// TIA Portal project "Project_MQTT" (V15.1)

(* hardware
DEVICE "S71500/ET200MP station_1"  S7-1500 station
   slot 0: "Rail_0"  Rack  6ES7 590-1***0-0AA0
   slot 1: "PLC_1"  CPU 1516F-3 PN/DP  6ES7 516-3FN01-0AB0  V2.6
      slot 3: "CPU display_1"  6ES7591-1BA00-0AA0
   slot 2: "TM Count 2x24V_1"  TM Count 2x24V  6ES7 550-1AA00-0AB0  V1.3
*)

// ===== PLC "PLC_1"  CPU 1516F-3 PN/DP =====

VAR_GLOBAL   // PLC tag table "Default tag table"
   "mxEnable" AT %M0.0 : Bool;
   "mxSaveIntoBroker" AT %M0.1 : Bool;
   "mxsubscribe" AT %M0.2 : Bool;
   "mxunsubscribe" AT %M0.3 : Bool;
   "mxPublishData" AT %M0.4 : Bool;
   "mxPublishData1" AT %M0.5 : Bool;
   "mxPublishData2" AT %M0.6 : Bool;
   "mxdone" AT %M0.7 : Bool;
   "Tag_1" AT %MW100 : Int;
END_VAR

// folder: 02_Types/S7-1500

TYPE "LMQTT_typePublishData"
   STRUCT
      publishMessage : Bool;   // Set to true. Can be reset to false once done flag is set be FB
      publishTopic : WString[250];   // Size be increased, but must increase MAX_SENDBUFFER and MAX_PUBLISH_MESSAGE in the FB
      publishMessageData : WString[1500];   // Size be increased, but must increase MAX_SENDBUFFER and MAX_PUBLISH_MESSAGE in the FB
      publishQoS : Int;   // Defines the QoS level for the MQTT message. 0,1 and 2 supported
      publishRetainFlag : Bool;   // If true, message may be saved at the broker
   END_STRUCT;
END_TYPE

TYPE "LMQTT_typeSubscribeData"
   STRUCT
      subscribeToTopic : Bool;   // When true, subscribes to the topic indicated by "subscriptionTopic"
      unsubscribeFromTopic : Bool;   // When true, unsubscribes from the "subscriptionTopic"
      subscriptionTopic : WString[250];   // Topic name to subscribe to or unsubscribe off
      subscriptionQoS : Int;   // Defines the QoS level for the MQTT message at the subscriber side. 0 and 1 allowed
   END_STRUCT;
END_TYPE

TYPE "LMQTT_typeSubscriptionData"
   STRUCT
      newMessageRecieved : Bool;   // Is TRUE for one cycle to signal that new data was recieved
      messageInvalid : Bool;   // Is TRUE, when either internal Buffer of FB is too small or recieved Message Data string length is too low
      receivingTopic : WString[400];   // The topic for which the message was recieved
      receivedMessageData : WString[2400];   // The received data (payload)
   END_STRUCT;
END_TYPE

TYPE "LMQTT_typeTcpConnParamData"
   STRUCT
      useQdn : Bool;   // When TRUE, configure the connection for TCP over the fully qualified domain name
      hwIdentifier : Hw_Any;   // HW_ID of the PROFINET interface of the CPU
      connectionID : Conn_Ouc;   // ID of the TCP connection
      qdnAdressBroker : String[254];   // URL of the MQTT Broker . Must end with a dot (".")
      ipAdressBroker : Array[0..3] of USInt;   // IP Address of the broker, e.g.: for the address "192.168.0.10"
      localPort : UInt := 0;   // Local port number of the CPU
      mqttPort : UInt := 1884;   // Remote port of the MQTT broker
      activateSecureConn : Bool;   // When TRUE, the communication is secured via TLS
      validateSubjectAlternateNameOfServer : Bool;   // Only relevant for Client side. If set to True, Client will validate IP address of broker against SAN in the certificate of the MQTT broker
      idTlsServerCertificate : UDInt;   // Identifier of X.509 certificate (usually a CA certificate) to validate the authetication of the TLS server. Only relevant, if "activateSecureConn" is "true"
      idTlsOwnCertificate : UDInt;   // Identifier of own X.509 certificate to validate the own authetication against the TLS server. Only relevant, if "activateSecureConn" is "true" and the TLS server requests a client authentication
   END_STRUCT;
   // // ipAdressBroker[0] : "192"
   // // ipAdressBroker[1] : "168"
   // // ipAdressBroker[2] : "0"
   // // ipAdressBroker[3] : "10"
END_TYPE

TYPE "LMQTT_typeParamData"
   STRUCT
      connectFlag : "LMQTT_typeConnectFlags";
      keepAlive : UInt := 30;   // can be set to higher or lower time // Default is 60 Seconds / KeepAlive in Seconds. 0=No Keepalive
      clientIdentifier : String[23] := 'Siemens SIMATIC';   // should be PROFINET devicename / Unique name of the client used from the client to identify itself at the broker during the connection establishment
      willTopic : String[100];   // specify topic where to send last will / If the will flag is set, the topic for the last will need to be defined
      willMessage : String[100];   // specify last will message which can be sent, see connect flags / If the will flag is set, the message for the last will needs to be defined
      userName : String[100];   // must be set, if flag "username" is true / If the username flag is set, the username for the login at the broker needs to be defined
      password : String[200];   // must be set, if flag "password" is true / If the password flag is set, the password for the login at the broker needs to be defined
   END_STRUCT;
END_TYPE

TYPE "LMQTT_typeConnectFlags"
   STRUCT
      cleanSession : Bool;   // if true, MQTT will create a clean Session at the Broker / When TRUE, all data from a previous session will be deleted
      will : Bool;   // if True, a last Will is sent when Mqtt Client (PLC) disconnects Broker / When TRUE, activates the last will and testament function
      willQoS1 : Bool;   // true, if QoS = 1 / When TRUE, the QoS has level 1 for the last will
      willQoS2 : Bool;   // true, if QoS = 2 / When TRUE, the QoS has level 2 for the last will
      willRetain : Bool;   // must be false, if Will flag is false / When TRUE, the last will is stored at the broker after its been sent
      password : Bool;   // if true, a password is required / When TRUE, the MQTT broker requires a login (name and password) of the client
      userName : Bool;   // if true, a username is required / When TRUE, the MQTT broker requires a login (name and password) of the client
   END_STRUCT;
END_TYPE

// folder: (top level)

DATA_BLOCK "LMQTT_Client_DB"   // DB1
{ S7_Optimized_Access := 'TRUE' }
AUTHOR : SiemensAG
FAMILY : MQTT
VERSION : 1.0
// stored: InstanceOfName LMQTT_Client
"LMQTT_Client"
BEGIN
END_DATA_BLOCK

DATA_BLOCK "db_publishData"   // DB2
{ S7_Optimized_Access := 'TRUE' }
VERSION : 0.1
BEGIN
   publishTopic := WSTRING#'drone/001';
END_DATA_BLOCK

DATA_BLOCK "db_subscribeData"   // DB3
{ S7_Optimized_Access := 'TRUE' }
VERSION : 0.1
BEGIN
END_DATA_BLOCK

DATA_BLOCK "db_tcpConnParam"   // DB4
{ S7_Optimized_Access := 'TRUE' }
VERSION : 0.1
BEGIN
   mqttPort := 1883;
   connectionID := 16#1;
   ipAdressBroker[0] := 192;
   ipAdressBroker[1] := 168;
   ipAdressBroker[2] := 11;
   ipAdressBroker[3] := 21;
   qdnAdressBroker := '192.168.11.21';
END_DATA_BLOCK

DATA_BLOCK "db_mqttParam"   // DB5
{ S7_Optimized_Access := 'TRUE' }
VERSION : 0.1
BEGIN
   willTopic := 'drone/001';
   willMessage := 'Sorry i am Died :(';
   connectFlag.will := True;
END_DATA_BLOCK

ORGANIZATION_BLOCK "Main"   // OB1, LAD, ProgramCycle
TITLE = "Main Program Sweep (Cycle)"
{ S7_Optimized_Access := 'TRUE' }
VERSION : 0.1
   VAR_INPUT
      Initial_Call : Bool;   // Initial call of this OB
      Remanence : Bool;   // =True, if remanent data are available
   END_VAR
   VAR CONSTANT
      cxAlwaysON : Bool := True;
   END_VAR
BEGIN

REGION Network 1: //
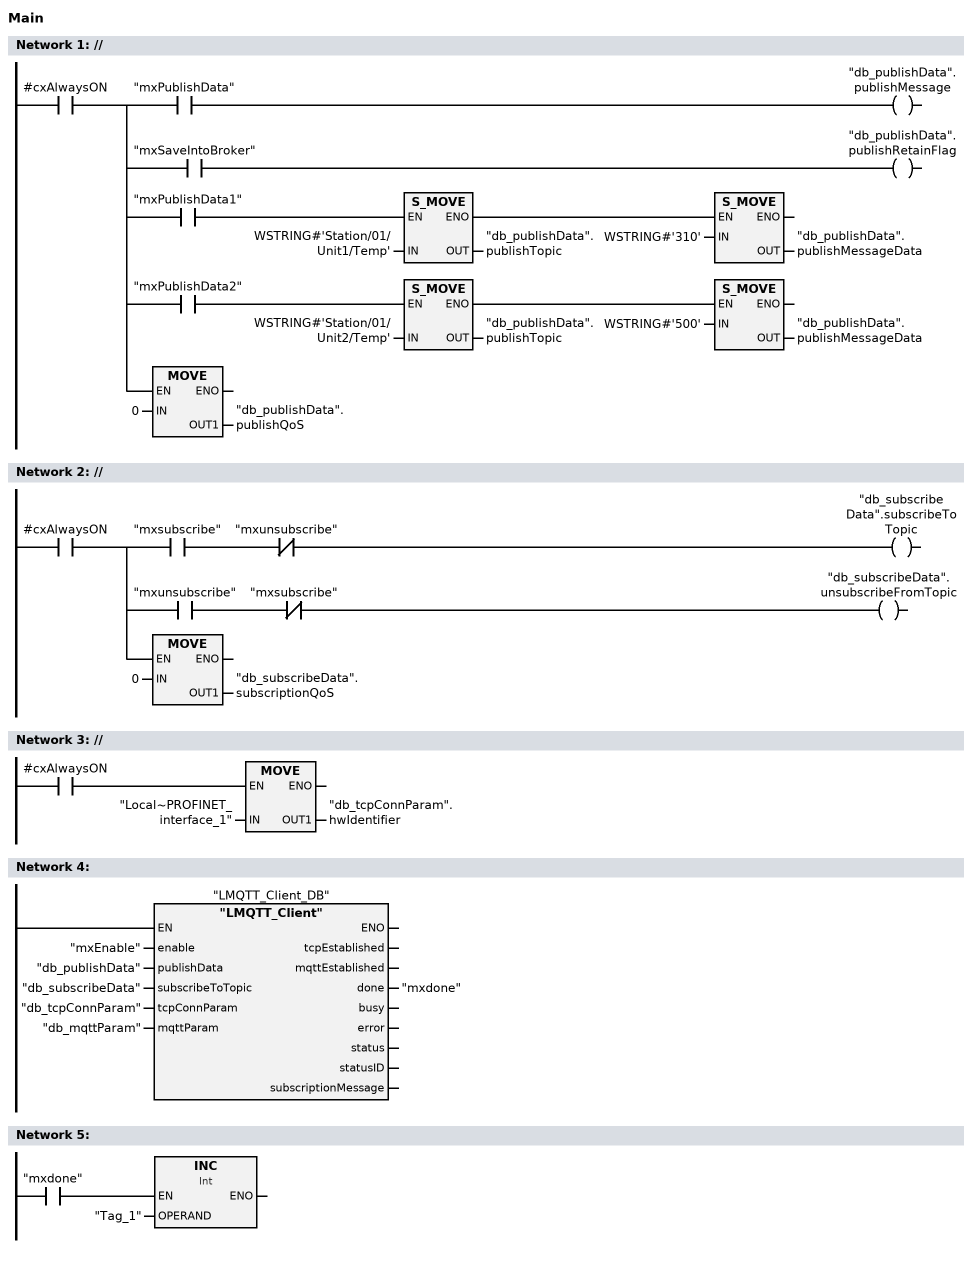
   RUNG wire#powerrail
      Contact( #cxAlwaysON )
      wire#w1
      Contact( "mxPublishData" )
      Coil( "db_publishData".publishMessage )
   END_RUNG
   RUNG wire#w1
      Contact( "mxSaveIntoBroker" )
      Coil( "db_publishData".publishRetainFlag )
   END_RUNG
   RUNG wire#w1
      Contact( "mxPublishData1" )
      S_Move(in := WSTRING#'Station/01/Unit1/Temp', out => "db_publishData".publishTopic)
      S_Move(in := WSTRING#'310', out => "db_publishData".publishMessageData)
   END_RUNG
   RUNG wire#w1
      Contact( "mxPublishData2" )
      S_Move(in := WSTRING#'Station/01/Unit2/Temp', out => "db_publishData".publishTopic)
      S_Move(in := WSTRING#'500', out => "db_publishData".publishMessageData)
   END_RUNG
   RUNG wire#w1
      Move(in := 0, out1 => "db_publishData".publishQoS)
   END_RUNG
   // the same network as SCL:
   "db_publishData".publishMessage := #cxAlwaysON AND "mxPublishData";
   "db_publishData".publishRetainFlag := #cxAlwaysON AND "mxSaveIntoBroker";
   IF #cxAlwaysON AND "mxPublishData1" THEN
       "db_publishData".publishTopic := WSTRING#'Station/01/Unit1/Temp';
       "db_publishData".publishMessageData := WSTRING#'310';
   END_IF;
   IF #cxAlwaysON AND "mxPublishData2" THEN
       "db_publishData".publishTopic := WSTRING#'Station/01/Unit2/Temp';
       "db_publishData".publishMessageData := WSTRING#'500';
   END_IF;
   IF #cxAlwaysON THEN "db_publishData".publishQoS := 0; END_IF;
END_REGION

REGION Network 2: //
   RUNG wire#powerrail
      Contact( #cxAlwaysON )
      wire#w1
      Contact( "mxsubscribe" )
      I_Contact( "mxunsubscribe" )
      Coil( "db_subscribeData".subscribeToTopic )
   END_RUNG
   RUNG wire#w1
      Contact( "mxunsubscribe" )
      I_Contact( "mxsubscribe" )
      Coil( "db_subscribeData".unsubscribeFromTopic )
   END_RUNG
   RUNG wire#w1
      Move(in := 0, out1 => "db_subscribeData".subscriptionQoS)
   END_RUNG
   // the same network as SCL:
   "db_subscribeData".subscribeToTopic := #cxAlwaysON AND "mxsubscribe" AND NOT "mxunsubscribe";
   "db_subscribeData".unsubscribeFromTopic := #cxAlwaysON AND "mxunsubscribe" AND NOT "mxsubscribe";
   IF #cxAlwaysON THEN "db_subscribeData".subscriptionQoS := 0; END_IF;
END_REGION

REGION Network 3: //
   RUNG wire#powerrail
      Contact( #cxAlwaysON )
      Move(in := "Local~PROFINET_interface_1", out1 => "db_tcpConnParam".hwIdentifier)
   END_RUNG
   // the same network as SCL:
   IF #cxAlwaysON THEN "db_tcpConnParam".hwIdentifier := "Local~PROFINET_interface_1"; END_IF;
END_REGION

REGION Network 4
   RUNG wire#powerrail
      "LMQTT_Client_DB"(enable := "mxEnable", publishData := "db_publishData", subscribeToTopic := "db_subscribeData", tcpConnParam := "db_tcpConnParam", mqttParam := "db_mqttParam", tcpEstablished =>, mqttEstablished =>, done => "mxdone", busy =>, error =>, status =>, statusID =>, subscriptionMessage =>)
   END_RUNG
   // the same network as SCL:
   "LMQTT_Client_DB"(enable := "mxEnable",   // "LMQTT_Client"
                     publishData := "db_publishData",
                     subscribeToTopic := "db_subscribeData",
                     tcpConnParam := "db_tcpConnParam",
                     mqttParam := "db_mqttParam",
                     done => "mxdone");
END_REGION

REGION Network 5
   RUNG wire#powerrail
      Contact( "mxdone" )
      { S7_Templates := "DestType := Int" } Inc( "Tag_1" )
   END_RUNG
   // the same network as SCL:
   IF "mxdone" THEN "Tag_1" := "Tag_1" + 1; END_IF;
END_REGION
END_ORGANIZATION_BLOCK

// folder: S7-1500

FUNCTION_BLOCK "LMQTT_Client"   // FB2, SCL
TITLE = LMQTT_Client
{ S7_Optimized_Access := 'TRUE' }
AUTHOR : SiemensAG
FAMILY : MQTT
VERSION : 1.0
   VAR_INPUT
      enable : Bool;   // Set TRUE, to establish a connection - set to FALSE to disconnect
      publishData : "LMQTT_typePublishData";   // Data area of MQTT publish message information
      subscribeToTopic : "LMQTT_typeSubscribeData";   // Data area of MQTT subscribe message information
      tcpConnParam : "LMQTT_typeTcpConnParamData";   // Data area of TCP connection information
      mqttParam : "LMQTT_typeParamData";   // Data area of MQTT connection
   END_VAR
   VAR_OUTPUT
      tcpEstablished : Bool;   // TRUE, if TCP connection established
      mqttEstablished : Bool;   // TRUE, if MQTT connection is established
      done : Bool;   // TRUE, if the job (connect, publish, subscribe) is successfully executed
      busy : Bool;   // TRUE, while the job is executed or a PING is being sent to the broker
      error : Bool;   // TRUE, if an error has occured
      status : DWord;   // Error message
      statusID : Int;   // State of the StateMachines where the error has occured
      subscriptionMessage : "LMQTT_typeSubscriptionData";   // Data area for receiving a message on a specific topic
   END_VAR
   VAR
      statTcpConnParam : TCON_IP_V4_SEC;   // Data area of TCP connection information
      statTcpConnParamQdn : TCON_QDN_SEC;   // Data area of TCP connection information over the fully qualified domain name
      instTcpConnect : TCON;   // Instance of the TCON function block
      instTcpSend : TSEND;   // Instance of the TSEND function block
      instTcpSendSubscribedMessagesAck : TSEND;   // Instance of the TSEND function block for Publish Ack
      instTcpRrcv : TRCV;   // Instance of the TRCV function block
      instTcpDisconnect : TDISCON;   // Instance of TDISCON function block
      instTconWatchDog : TON_TIME;   // Set watchdog time for TCP Connection
      instTrcvWatchDogTimeout : TON_TIME;   // Set watchdog time for receiving data over an existing communication connection
      instMqttKeepAlivePing : TON_TIME;   // Set the MQTT KeepAlive Timer
      instMqttAcknowledgeWatchDog : TON_TIME;   // Set watchdog time for MQTT CONACK Packet
      statStateTcpMachine : Int;   // Current state for TCP state machine
      statStateTrcvMachine : Int := 40;   // Current state for TRCV state machine
      statStateMqttMachine : Int;   // Current state for MQTT state machine
      statStateMqttJobMachine : Int;   // Current state for the MQTT Job (publish/subscribe/unsubscribe)
      statSwitchCaseHeaderType : Int;   // Current header type based on packet type (CONACK, PUBACK, ...)
      statLastState : Int;   // Saves the last state of a specific job in case of error
      statConnectLength : Int;   // Length in bytes of the MQTT connect packet
      statCorrectOffset : Int;   // Static variable used for building the telegram in case "Last Will and Testament" activated
      statSendLength : Int;   // Length of the packet to be sent to the broker
      statConnectEncodedLength : Int;   // Length of the MQTT connect packet encoded
      statConnectLengthOffset : Int;   // Static variable used for building the telegram, step by step
      statMqttKeepAliveTime : Time;   // Duration of the MQTT keep alive time, the longest period of time that the broker and client can endure without sending a message
      statCnt : DInt;   // Static variable for counting the bytes for further processings
      statCntOffset : Int;   // Static variable to count the remaining length pf packet
      statPacketID : Int;   // Packet identifier which uniquely identifies a message between client and broker. Only relevant ofr QoS>0
      statPacketIDAck : Int;   // Static variable used to check if the PacketID of the Publish packet matches the received Puback packet
      statPublishOld : Bool;   // Last cycle's value of input "publishData.publishMessage"
      statEnableOld : Bool;   // Last cycle's value of input "enable"
      statEnableTconWatchDogTimer : Bool;   // Start watchdog timer for TCON
      statEnableTrcvWatchDogTimer : Bool;   // Start watchdog timer for TRCV
      statEnableMqttKeepAliveTimer : Bool;   // Start keep alive timer for MQTT
      statEnableMqttAckWatchDog : Bool;   // Start watchdog timer for MQTT CONACK packet
      statMqttKeepAliveOff : Bool;   // Static variable used when no Keep Alive timer was set
      statRemainingLenOfRecMessage : UDInt;   // The total remaining length to be expected of the packet according to data package header provided
      statSendBuffer : Array[1..#MAX_SENDBUFFER] of Byte;   // can be changed, Must be atleast len of Topic + Len of Msg when publishing / Buffer for sending the published data
      statSendBufferSubscribePacketAckn : Array[1..20] of Byte;   // do not change / Buffer for sending the publish acknowledgement packet
      statTrcvMessageBuffer : Array[1..#MAX_TRCV_1400] of Byte;   // do not change / Buffer for receiving the data for the topic to which we have subscribed
      statTrcvHeaderBuffer : Array[1..5] of Byte;   // do not change / Buffer for the MQTT Header
      statInternalBodyBuffer : Array[1..#MAX_INTERNAL_BUFFERLEN] of Byte;   // can be changed, Must be atleast len of Topic + Len of Msg when subscribing / Buffer for the received messages
      statSubscribeOld : Bool;   // Last cycle's value of input "subscribeToTopic.subscribeToTopic"
      statUnsubcribeOld : Bool;   // Last cycle's value of input "subscribeToTopic.unsubscribeFromTopic"
      statStateMqttReceive : Int;   // State of the MQTT procedure based on QoS
      statPacketID2 : Word;   // PacketID used for sending a PUBACK in case we subscribed on a topic with QoS=1
      statPubPacEncoded : Bool;   // TRUE, when data is encoded and when TRUE start sending the data
      statSubPacEncoded : Bool;   // TRUE, when subscribe request packet is encoded and when TRUE then the subscribe request packet is sent to the broker
      statUnsubPacEncoded : Bool;   // TRUE, when unsubscribe request packet is encoded and when TRUE then the unsubscribe request packet is sent to the broker
      statQoS1decoded : Bool;   // TRUE, when received topic/message with QoS=1 was succesfully decoded
      statPingPacEncoded : Bool;   // TRUE, when PING packet is encoded and when TRUE then the PING request packet is sent to the broker
      statTrcvlen : UDInt;   // Amount of received data in bytes
      statInternalBufferCount : DInt;   // Counts the bytes of the internal buffer
      statInternalBufferOverflow : Bool;   // TRUE when the received message on a topic we subscribed to is bigger than the internal buffer
      statRecPackageQoSsaver : Int;   // Static variable used to store information on QoS for later use
      statTotalRemainingMessageLengthSaver : UDInt;   // Static variable used to save the remaining length of recieved package for later use
      statStringToCharBuffer : Array[0..#MAX_USER_PW_WILL_LEN] of Char;   // should be greater than username or password string / Buffer for transforming ClientIdentifier, Will, Username, Password from string to char
      statWStringToWCharBuffer : Array[0..#MAX_PUBLISH_MESSAGE] of WChar;   // should be greater than topic or payload size to be published / Buffer for transforming the publishTopic and publishMessageData from wstring to wchar
      statDisconnect : Bool;   // Will be true if FB has to disconnect
      statBusy : Bool;   // TRUE when FB is busy
      statDone : Bool;   // TRUE, if the job (connect, publish, subscribe) is successfully executed
      statError : Bool;   // TRUE, if an error has occured
      statStatus : DWord;   // Error message
      statStatusID : Int;   // State of the StateMachines where the error has occured
      statTcpEstablished : Bool;   // TRUE, if TCP connection established
      statMqttEstablished : Bool;   // TRUE, if MQTT connection is established
   END_VAR
   VAR_TEMP
      tempCountChars : UInt;   // Used for the conversion from string to CHAR to count the number of characters
      tempWordForSliceAddress : Word;   // Temporary variable just used for the conversion from UINT to WORD for slice addressing
      tempMultiplier : UDInt;   // Temporary variable used in the algorithm for decoding the remaining length field
      tempLength : Word;   // Temporary variable just used for the conversion from INT to WORD for slice addressing
      tempCnt : DInt;   // Temporary variable used for iterating among different received data lenghs
      tempReceivedMessage : Bool;   // TRUE when received message on subscription
      tempRecPubTopicLength : UInt;   // The length of the topic for which the message was received (through subscription)
      tempPubRec : Bool;   // TRUE, if the received packet is a PUBREC packet. Relevant for QoS=2
      tempPubAck : Bool;   // TRUE, if the received packet is a PUBACK packet
      tempConAck : Bool;   // TRUE, if the received packet is a CONNACK packet
      tempPingResp : Bool;   // TRUE, if the received packet is a PINGRESP packet
      tempPubComp : Bool;   // TRUE, if the received packet is a PUBCOMP packet
      tempSubAck : Bool;   // TRUE, if the received packet is a SUBACK packet
      tempUnSubAck : Bool;   // TRUE, if the received packet is a UNSUBACK packet
   END_VAR
   VAR CONSTANT
      MAX_INTERNAL_BUFFERLEN : UDInt := 3000;   // Maximum buffer length for the received messages in bytes
      MAX_TRCV_1400 : UDInt := 1400;   // Maximum amount of received data in bytes in one cycle
      MAX_SENDBUFFER : Int := 2000;   // Maximum amount of send buffer in bytes; Must be the size of Topic Len + Message Len
      MAX_USER_PW_WILL_LEN : Int := 250;   // Maximum length of the buffer to store Username, Passwort, Will Topic and Will message in bytes
      MAX_PUBLISH_MESSAGE : Int := 1550;   // Maximum length of the published message in bytes
      EMPTY : WString;   // Empty string
      EMPTY_CHAR : Char := ' ';   // Empty Char
      EMPTY_WCHAR : WChar := WCHAR#' ';   // Empty WChar
      TOPIC_LEN_INFO : UInt := 2;   // According to MQTT, 2 byte are allocated for the topic length information
      DEFAULT_PACKET_ID : Int := 10;   // Set a default value for the PacketID
      TRCV_WAIT_FOR_HEADER : Int := 40;   // First step of TRCV StateMachine
      TRCV_WAIT_FOR_BODY : Int := 48;   // Second step of TRCV StateMachine, after receiving the header of the package we wait for the body
      TCP_PARAM : Int := 1;   // First step of the TCP StateMachine - initializing the TCP connection parameters
      TCP_DISCONNECT : Int := -1;   // Disconnected state of the TCP StateMachine
      TCP_ERROR : Int := -2;   // Error state of TCP StateMachine
      TCP_CONNECTED : Int := 3;   // Connected state of TCP StateMachine
      TCP_CONNECTING : Int := 2;   // After TCP parameters initialization, go to connecting state = set the rising edge for TCON
      MQTT_DISCONNECT_STATE : Int := 9;   // State in which the DISCONNECT MQTT packet is built and sent
      MQTT_CONNECT_FLAG_CHECK_STATE : Int := 10;   // MQTT state in which the correctness of the flags is checked
      MQTT_CONNECT_STATE : Int := 11;   // After checking that the flags are correctly set, go to Connect state of the MQTT StateMachine and form the MQTT CONNECT packet and after that try to connect to the broker
      MQTT_CONNACK_STATE : Int := 12;   // After CONNECT packet was send wait for the CONNACK packet (#tempConAck) to be received
      MQTT_PUBLISH_STATE : Int := 13;   // State in which a PUBLISH packet is sent
      MQTT_PUBLISH_EVAL_STATE : Int := 24;   // State which evaluates if a PUBLISH packet with QoS=0 was successful
      MQTT_PUBACK_STATE : Int := 14;   // State which evaluates if a PUBLISH packet with QoS=1 was successful
      MQTT_SUBSCRIBE_STATE : Int := 15;   // State in which the SUBSCRIBE packet is processed and the subscription on a specific topic is performed
      MQTT_CONNECTED_STATE : Int := 16;   // Connected state of the MQTT StateMachine - if the CONNACK was successfully received
      MQTT_UNSUBSCRIBE_STATE : Int := 22;   // State in which the UNSUBSCRIBE packet is processed and the unsubscription from a specific topic is performed
      MQTT_UNSUBACK_STATE : Int := 23;   // State in which the UNSUBACK packet is evaluated
      MQTT_SUBACK_STATE : Int := 21;   // State in which the SUBACK packet is evaluated
      MQTT_PING : Int := 17;   // State in which PINGREQ packet is formed and sent
      MQTT_PINGRESP : Int := 18;   // State in which the PINKRESP packet is received and evaluated
      MQTT_PUBREC_ACK_STATE : Int := 19;   // State which evaluates if a PUBLISH packet with QoS=2 was acknowledged by the broker
      MQTT_PUBCOMP_STATE : Int := 20;   // State which evaluates if a PUBREL packet with QoS=2was successful
      MQTT_PUBREC_SEND_STATE : Int := 29;   // State which sends the PUBREL packet as response to the received PUBREC packet, for QoS=2
      MQTT_RECEIVED_QOS0_STATE : Int := 25;   // State in which we decode a message recevived with a QoS=0
      MQTT_RECEIVED_QOS1_STATE : Int := 26;   // State in which we decode a message recevived with a QoS=1
      MQTT_RECEIVED_QOS2_STATE : Int := 27;   // NOT IMPLEMENTED
      MQTT_DISCONNECTED_STATE : Int := -11;   // Disconnected state of MQTT StateMachine
      MQTT_ERROR_STATE : Int := -12;   // Error state of the MQTT StateMachine
      MQTT_TIMEOUT_ID : Int := -13;   // State which signals that the keepalive was triggered but there was no reaction from server within keep alive timer
      MQTT_BAD_ID : Int := -14;   // State which signals that the remaining length of the CONNACK packet is different than 2
      MQTT_QOS_MISMATCH_ID : Int := -15;   // State which signals that the requested QoS does not match the granted QoS in the SUBACK packet
      IDLE : Int := 0;   // State in which no job is performed
      TIME_MONITORING_ID : Int := -16;   // State which occurs when the watchon time for establishing a TCP connection was exceeded
      TCON_WATCHDOG_TIME : Time := t#30s;   // Watchdog Timer for establishing a connection
      TRCV_WATCHDOG_TIME : Time := T#15s;   // Watchdog Timer for receiving subscribed data from a broker. may be set to a higher limit on slow internet connections
      MQTT_ACK_WATCHDOG_TIME : Time := t#10s;   // Watchdog Timer for recieving a MQTT Response telegram from a broker
      MQTT_CONACK_FLAG_SP : Int := 1;   // Connect acknowledge flag in case no Session Present flag was set
      MQTT_MSG_TYPE_CONNECT : Int := 16;   // CONNECT MQTT Control Packet (see MQTT standard for more info)
      MQTT_MSG_TYPE_CONNACK : Int := 32;   // CONNACK MQTT Control Packet (see MQTT standard for more info)
      MQTT_MSG_TYPE_DISCONNECT : Int := 224;   // DISCONNECT MQTT Control Packet (see MQTT standard for more info)
      MQTT_MSG_TYPE_PUBACK : Int := 64;   // PUBACK MQTT Control Packet (see MQTT standard for more info)
      MQTT_MSG_TYPE_PUBREL : Int := 98;   // PUBREL MQTT Control Packet (see MQTT standard for more info)
      MQTT_MSG_TYPE_PUBREC : Int := 80;   // PUBREC MQTT Control Packet (see MQTT standard for more info)
      MQTT_MSG_TYPE_PUBCOM : Int := 112;   // PUBCOM MQTT Control Packet (see MQTT standard for more info)
      MQTT_MSG_TYPE_SUBSCRIBE : Int := 130;   // SUBSCRIBE MQTT Control Packet (see MQTT standard for more info)
      MQTT_MSG_TYPE_UNSUBSCRIBE : Int := 162;   // UNSUBSCRIBE MQTT Control Packet (see MQTT standard for more info)
      MQTT_MSG_TYPE_SUBACK : Int := 144;   // SUBACK MQTT Control Packet (see MQTT standard for more info)
      MQTT_MSG_TYPE_UNSUBACK : Int := 176;   // UNSUBACK MQTT Control Packet (see MQTT standard for more info)
      MQTT_MSG_TYPE_PING : Int := 192;   // PING MQTT Control Packet (see MQTT standard for more info)
      MQTT_MSG_TYPE_PINGRESP : Int := 208;   // PINGRESP MQTT Control Packet (see MQTT standard for more info)
      MQTT_MSG_TYPE_PUB_INC_MESSAGE_QoS0 : Int := 48;   // PUBLISH MQTT Control Packet for QoS = 0 (see MQTT standard for more info)
      MQTT_MSG_TYPE_PUB_INC_MESSAGE_QoS1 : Int := 50;   // PUBLISH MQTT Control Packet for QoS = 1 (see MQTT standard for more info)
      MQTT_MSG_TYPE_PUB_INC_MESSAGE_QoS2 : Int := 52;   // PUBLISH MQTT Control Packet for QoS = 2 (see MQTT standard for more info)
      MQTT_MSG_TYPE_PUB_INC_MESSAGE_BAD : Int := 54;   // PUBLISH MQTT Control Packet for QoS =1 and QoS=2 at the same time (see MQTT standard for more info)
      MQTT_CONNACK_ACCEPTED : Int := 0;   // Connect acknowledge flag in case no session present flag was not set
      MQTT_ERROR_BADMESSAGE : Word := 16#80F6;   // Error occurs when we receive a message that has QoS=1 and QoS=2 at the sime time
      MQTT_ERROR_WILL_FLAG : Word := 16#80F0;   // Error occurs when the willRetain flag ist set true without setting the Will flag to true
      MQTT_ERROR_QOS_FLAG : Word := 16#80F1;   // Error occurs when the QoS of the Will is set without setting the Will flag to true or it accurs when the QoS=1 and 2 at the same time
      MQTT_ERROR_PACKETID : Word := 16#80F2;   // Error occurs when the acknowledge failes ( the packet ID of the acknowledgement packet does not match the original packet ID)
      MQTT_ERROR_KEEPALIVE : Word := 16#80F3;   // Error occurs when the Keep Alive time is set to 1 or 2 seconds
      MQTT_ERROR_QOS_MISMATCH : Word := 16#80F4;   // Error occurs when we try to publish a message with a QoS < 0 and a QoS > 2
      MQTT_ERROR_TOPIC_EMPTY : Word := 16#80F5;   // Error occurs when we try to publish/subscribe to an empty topic
      MQTT_ERROR_SUBSCRIPTION_FAILURE : Word := 16#80F7;   // Error occurs by subcription when the return code of the SUBACK Packet from the Broker containts a Failure
      TCP_TRCV_COMMUNICATION_ERROR : Word := 16#80C0;   // Any TRCV error that is related to a Communication Issue
      TCON_ERROR_CONID_IN_USE : Word := 16#80A3;   // CON ID is in use
      BIT_MASK_HIGHBITS : Word := 16#F0;   // MQTT Message Types only use High bits, so we only use High bits and ignore low bits
      BIT_MASK_LOWBITS : Word := 16#0F;   // MQTT Message Types only use Low bits, so we only use low bits and ignore high bits
      BIT_MASK_ALL : Word := 16#FF;   // MQTT Message Type that uses all bits
      BIT_MASK_QOS : Word := 16#F6;   // A Bit Mask to only validate recieved Byte against QOS Value
      DEFAULT_VALUE_ZERO : Int := 0;   // DEFAULT Value for Variables that a ZERO Based
      QOS_0 : Int := 0;   // Set to QoS0
      QOS_1 : Int := 1;   // Set to QoS1
      QOS_2 : Int := 2;   // Set to QoS2
      CONST_128_CALC : Int := 128;   // Default mulitplier to calculate package length
      MQTT_PROTOCOL_LEVEL : Int := 4;   // MQTT Protocol Level 4 = Version Mqtt 3.1
      DEFAULT_TWO_BYTE_LEN : Int := 2;   // When building Telegram, adds 2 byte for each parameter to the total package length
      DEFAULT_THREE_BYTE_LEN : Int := 3;   // Default Value for 3 Bytes
      MAX_INT : Int := 32767;   // Max Value of a UINT
   END_VAR
   // statTcpConnParamQdn.ConnPara.ID := 16#6;
   // statTcpConnParam.ConnPara.ConnectionType := 16#B;
   // statTcpConnParam.ConnPara.ActiveEstablished := 1;
   // statTcpConnParam.ConnPara.ID := 16#6;
   // statTcpConnParamQdn.ConnPara.ConnectionType := 16#0B;
   // statTcpConnParamQdn.ConnPara.ActiveEstablished := 1;
   // // mqttParam.connectFlag : Data area of MQTT connection flags
   // // instTconWatchDog.IN : When TRUE, start the timer
   // // instTconWatchDog.Q : TRUE, if the "PT" duration has expired
   // // instTconWatchDog.PT : Duration of the delay/watchdog timer
   // // instTconWatchDog.ET : Current timer value
   // // instTrcvWatchDogTimeout.Q : TRUE, if the "PT" duration has expired
   // // instTrcvWatchDogTimeout.IN : When TRUE, start the timer
   // // instTrcvWatchDogTimeout.ET : Current timer value
   // // instTrcvWatchDogTimeout.PT : Duration of the delay/watchdog timer
   // // instMqttKeepAlivePing.PT : Duration of the delay/KeepAlive timer
   // // instMqttKeepAlivePing.ET : Current timer value
   // // instMqttKeepAlivePing.IN : When TRUE, start the timer
   // // instMqttKeepAlivePing.Q : TRUE, if the "PT" duration has expired
   // // instMqttAcknowledgeWatchDog.PT : Duration of the delay/watchdog timer
   // // instMqttAcknowledgeWatchDog.ET : Current timer value
   // // instMqttAcknowledgeWatchDog.IN : When TRUE, start the timer
   // // instMqttAcknowledgeWatchDog.Q : TRUE, if the "PT" duration has expired
BEGIN
   REGION Header
       //=============================================================================
       //SIEMENES AG
       //(c)Copyright 2019 All Rights Reserved
       //-----------------------------------------------------------------------------
       //Library:       LMqtt_Client
       //Tested with:   S7-1516 FW V2.6.1
       //Engineering:   TIA Portal V15.1
       //Restrictions:  -
       //Requirements:  At least CPU Firmware V 2.1
       //Functionality: MQTT Client
       //-----------------------------------------------------------------------------
       //Change log table:
       //Version  Date       Expert in charge              Changes applied
       //01.00.00 06.06.2017 Siemens Online Support        First released version
       //02.00.00 04.06.2018 DF FA S SUP E&C (COM)         Added DNS support and Subscribe to topics
       //02.01.00 10.11.2019 DF FA S SUP E&C (COM)         Minor connection improvements. Updated some Comments
       //02.01.01 16.03.2020 DF FA S SUP E&C (COM)         Fixed Issue with SAN Bit not setting correct.
       //=============================================================================

   END_REGION

   REGION First Execute/Rising Edge
       IF #enable // Only executed on first trigger / Rising edge
           AND NOT #statEnableOld
       THEN
           #statLastState := #IDLE;
           #statStateTcpMachine := #TCP_PARAM; //first step of TCP StateMachine
           #statStateMqttMachine := #MQTT_DISCONNECTED_STATE; //first step of MQTT StateMachine
           #statStateTrcvMachine := #TRCV_WAIT_FOR_HEADER;//first step of TRCV StateMachine

           #statTcpConnParam.ConnPara.ID := #tcpConnParam.connectionID;
           #statTrcvlen := 0;
           #statRemainingLenOfRecMessage := 0;
           #statTotalRemainingMessageLengthSaver := 0;
           #statEnableTconWatchDogTimer := false; //Reset Watchdog
           #statEnableTrcvWatchDogTimer := FALSE;
           #statEnableMqttKeepAliveTimer := FALSE;
           #statPublishOld := #publishData.publishMessage;
           #statSubscribeOld := #subscribeToTopic.subscribeToTopic;
           #statUnsubcribeOld := #subscribeToTopic.unsubscribeFromTopic;
           #statError := false;
           #statDisconnect := false;
           #statStatus := 0;
           #statStatusID := 0;
       END_IF;
   END_REGION

   REGION Last Execute / Falling edge
       IF NOT #enable // falling edge of enable
           AND #statEnableOld
       THEN
           IF #statError = true // if falling edge and error is persistent
           THEN
               #statStateTcpMachine := #TCP_DISCONNECT;
               #statError := false;
           ELSE // if falling edge and no error is persistent, try mqtt disconnect then disconnect TCP.
               #statStateMqttMachine := #MQTT_DISCONNECT_STATE;
               //#statStateTCP := #TCP_DISCONNECT; Is done in MQTT Disconnect
           END_IF;
       END_IF;
   END_REGION

   REGION WATCHDOG TIMER TCP
       //Start watchdog timer for TCON and TRCV
       #instTconWatchDog(IN := #statEnableTconWatchDogTimer,
                         PT := #TCON_WATCHDOG_TIME);//default is 30 Seconds

       #instTrcvWatchDogTimeout(IN := #statEnableTrcvWatchDogTimer,
                                PT := #TRCV_WATCHDOG_TIME);//default is 15 seconds
   END_REGION

   REGION State machine TCP
       CASE #statStateTcpMachine OF
           #IDLE:
               REGION IDLE
                   //In IDLE we wont try to do MQTT Connect, as TCP is not connected.
                   IF NOT #statError
                   THEN
                       //Default outputs, signal fb is ready.
                       #statStatus := 0;
                       #statStatusID := 0;
                       #statError := 0;
                       #statTcpEstablished := false;
                       #statMqttEstablished := false;


                       #subscriptionMessage.newMessageRecieved := FALSE;
                       #subscriptionMessage.receivedMessageData := #EMPTY;
                       #subscriptionMessage.receivingTopic := #EMPTY;

                       #statTcpConnParam.ConnPara.ID := #tcpConnParam.connectionID;
                       //Finish tdiscon in defined State;
                       #instTcpDisconnect(ID := #statTcpConnParam.ConnPara.ID);
                       //Finish TRCV call in defined State
                       IF #instTcpRrcv.STATUS <> 16#80A1 // connection has not yet been established or is terminated.
                       THEN
                           #instTcpRrcv(EN_R := true,
                                        ID := #statTcpConnParam.ConnPara.ID,
                                        LEN := 0,
                                        ADHOC := 1,
                                        DATA := #statTrcvHeaderBuffer);
                       END_IF;

                       IF #tcpConnParam.useQdn
                       THEN //finish call of TCON in defined state, but no .req is issued.
                           #instTcpConnect(ID := #statTcpConnParam.ConnPara.ID,
                                           CONNECT := #statTcpConnParamQdn);
                       ELSE
                           #instTcpConnect(ID := #statTcpConnParam.ConnPara.ID,
                                           CONNECT := #statTcpConnParam);
                       END_IF;
                   END_IF;

                   // IF error occured:

                   #statDone := false;
                   #statBusy := false;
                   #statMqttEstablished := false;
                   #statTcpEstablished := false;
                   #statStateMqttMachine := #MQTT_DISCONNECTED_STATE;
                   #statEnableTconWatchDogTimer := false;
                   #statEnableTrcvWatchDogTimer := FALSE;
                   #statEnableMqttKeepAliveTimer := false;
                   #statEnableMqttAckWatchDog := FALSE;

                   IF #statLastState = #TCP_DISCONNECT
                   THEN
                       #statError := FALSE;
                   END_IF;

               END_REGION

           #TCP_PARAM:
               REGION TCP Param 
                   //assign TCON Params here

                   IF #tcpConnParam.useQdn THEN

                       #statTcpConnParamQdn.ConnPara.InterfaceId := #tcpConnParam.hwIdentifier;
                       #statTcpConnParamQdn.ConnPara.ID := #tcpConnParam.connectionID;
                       #statTcpConnParamQdn.ConnPara.LocalPort := #tcpConnParam.localPort;
                       #statTcpConnParamQdn.ConnPara.RemotePort := #tcpConnParam.mqttPort;
                       #statTcpConnParamQdn.ConnPara.RemoteQDN := #tcpConnParam.qdnAdressBroker;
                       #statTcpConnParamQdn.ActivateSecureConn := #tcpConnParam.activateSecureConn;
                       #statTcpConnParamQdn.TLSClientCertRef := #tcpConnParam.idTlsOwnCertificate;
                       #statTcpConnParamQdn.TLSServerCertRef := #tcpConnParam.idTlsServerCertificate;
                       #statTcpConnParamQdn.ExtTLSCapabilities.%X0 := #tcpConnParam.validateSubjectAlternateNameOfServer;
                   ELSE
                       #statTcpConnParam.ConnPara.InterfaceId := #tcpConnParam.hwIdentifier;
                       #statTcpConnParam.ConnPara.ID := #tcpConnParam.connectionID;
                       #statTcpConnParam.ConnPara.LocalPort := #tcpConnParam.localPort;
                       #statTcpConnParam.ConnPara.RemotePort := #tcpConnParam.mqttPort;
                       #statTcpConnParam.ConnPara.RemoteAddress.ADDR[1] := USINT_TO_BYTE(#tcpConnParam.ipAdressBroker[0]);
                       #statTcpConnParam.ConnPara.RemoteAddress.ADDR[2] := USINT_TO_BYTE(#tcpConnParam.ipAdressBroker[1]);
                       #statTcpConnParam.ConnPara.RemoteAddress.ADDR[3] := USINT_TO_BYTE(#tcpConnParam.ipAdressBroker[2]);
                       #statTcpConnParam.ConnPara.RemoteAddress.ADDR[4] := USINT_TO_BYTE(#tcpConnParam.ipAdressBroker[3]);
                       #statTcpConnParam.ActivateSecureConn := #tcpConnParam.activateSecureConn;
                       #statTcpConnParam.TLSClientCertRef := #tcpConnParam.idTlsOwnCertificate;
                       #statTcpConnParam.TLSServerCertRef := #tcpConnParam.idTlsServerCertificate;
                       #statTcpConnParam.ExtTLSCapabilities.%X0 := #tcpConnParam.validateSubjectAlternateNameOfServer;

                   END_IF;

                   //move on to TCON Init
                   #statStateTcpMachine := #TCP_CONNECTING;
               END_REGION

           #TCP_CONNECTING:
               REGION TCP Connecting
                   //Start watchdog timer
                   #statEnableTconWatchDogTimer := true;

                   //Set rising edge for TCON:
                   #instTcpConnect.REQ := NOT #instTcpConnect.REQ XOR #instTcpConnect.BUSY;

                   #statBusy := true;
                   //CALL TCON Instance
                   //
                   IF #tcpConnParam.useQdn
                   THEN
                       #instTcpConnect(ID := #statTcpConnParam.ConnPara.ID,
                                       CONNECT := #statTcpConnParamQdn);
                   ELSE
                       #instTcpConnect(ID := #statTcpConnParam.ConnPara.ID,
                                       CONNECT := #statTcpConnParam);
                   END_IF;


                   IF (#instTcpConnect.DONE)
                       AND (#instTcpConnect.BUSY = false)
                       AND (#instTcpConnect.REQ)
                   THEN
                       // #statBusy := false;
                       #instTcpConnect.REQ := false;
                       #statTcpEstablished := true;
                       #statStateTcpMachine := #TCP_CONNECTED; // go to Connected Step
                       #statEnableTconWatchDogTimer := false; //RESET Watchdog
                   ELSIF #instTcpConnect.ERROR
                   THEN
                       #statStatusID := #TCP_CONNECTING;
                       #instTcpConnect.REQ := false;
                       #statStateTcpMachine := #TCP_ERROR;
                       #statLastState := #TCP_DISCONNECT;

                       // WatchDog FOR TCON Connection was triggered
                   ELSIF (#instTconWatchDog.Q = true)  //Default watchdog Time is 30 sec
                   THEN//in next cycle, switch from TCP Connecting to TCP Error State
                       #instTcpConnect.REQ := false;
                       #statStateTcpMachine := #TCP_ERROR;
                       #statStatusID := #TIME_MONITORING_ID;
                   END_IF;

               END_REGION
           #TCP_CONNECTED:
               REGION TCP Connected
                   //Only when connected, TSEND and TRCV make sense
                   REGION CALL OUC TSEND/TRCV blocks    

                       //always execute Send and Recieve
                       #instTcpSend(ID := #statTcpConnParam.ConnPara.ID,
                                    DATA := #statSendBuffer);
                       #instTcpSendSubscribedMessagesAck(ID := #statTcpConnParam.ConnPara.ID,
                                                         DATA := #statSendBufferSubscribePacketAckn);

                       IF #statStateTrcvMachine = #TRCV_WAIT_FOR_HEADER //decide, if header or body recieve area
                       THEN
                           //recieve header
                           #instTcpRrcv(EN_R := true,
                                        ID := #statTcpConnParam.ConnPara.ID,
                                        LEN := 0,
                                        ADHOC := 1,
                                        DATA := #statTrcvHeaderBuffer); //recieves up to 5 byte  
                       ELSIF #statStateTrcvMachine = #TRCV_WAIT_FOR_BODY
                       THEN
                           //recieve body
                           #instTcpRrcv(EN_R := true,
                                        ID := #statTcpConnParam.ConnPara.ID,
                                        LEN := #statTrcvlen,
                                        ADHOC := 0,
                                        DATA := #statTrcvMessageBuffer);

                           //might add generic error ELSE here
                       END_IF;

                   END_REGION

                   //Check TCP Connection
                   IF #instTcpRrcv.STATUS > #TCP_TRCV_COMMUNICATION_ERROR //If Status occured, TCP not ok
                   THEN
                       //TCP Is in error, we go to Disconnect and then Error 
                       #statDisconnect := TRUE;
                       #statStatus := #instTcpRrcv.STATUS;
                       #statStateTcpMachine := #TCP_DISCONNECT;
                       #statStatusID := #TCP_CONNECTED;
                   ELSE // TCP IS OK Execute data evaluation
                       REGION TCP OK, WAIT for TRCV in a StateMachine                       
                           //SO we wait in Wait_for_Header State, until header was recieved. then we evaluate and handle.
                           CASE #statStateTrcvMachine OF
                               #TRCV_WAIT_FOR_HEADER:  // Statement Case Wait for Header Pakets
                                   REGION WAIT FOR HEADER
                                       // Wait for TRCV to complete and new data rising edge
                                       #statSwitchCaseHeaderType := #DEFAULT_VALUE_ZERO; // bring inside state to default

                                       IF #instTcpRrcv.BUSY = false AND #instTcpRrcv.NDR = TRUE
                                       THEN
                                           //consistent 5 byte in buffer,check HeaderIdentifier
                                           #statSwitchCaseHeaderType := WORD_TO_INT((#statTrcvHeaderBuffer[1] AND #BIT_MASK_HIGHBITS));
                                           REGION Act on MsgType                                        
                                               CASE #statSwitchCaseHeaderType OF
                                                   #MQTT_MSG_TYPE_CONNACK:  // When its CONNACK Packet
                                                       REGION CONACK_PACKET                                                    
                                                           #tempConAck := TRUE; //We will evaluate in MQTT StateMachine Below the response
                                                           #statSwitchCaseHeaderType := #DEFAULT_VALUE_ZERO;
                                                       END_REGION
                                                   #MQTT_MSG_TYPE_PUBACK:
                                                       REGION PUBACK_PACKET  
                                                           #tempPubAck := TRUE;
                                                           #statSwitchCaseHeaderType := #DEFAULT_VALUE_ZERO;
                                                       END_REGION
                                                   #MQTT_MSG_TYPE_PUBREC:
                                                       REGION PUBREC_PACKET  
                                                           #tempPubRec := TRUE;
                                                           #statSwitchCaseHeaderType := #DEFAULT_VALUE_ZERO;
                                                       END_REGION
                                                   #MQTT_MSG_TYPE_PUBCOM:
                                                       REGION PUBCOMP_PACKET  
                                                           #tempPubComp := TRUE;
                                                           #statSwitchCaseHeaderType := #DEFAULT_VALUE_ZERO;
                                                       END_REGION
                                                   #MQTT_MSG_TYPE_SUBACK:
                                                       REGION SUBACK_PACKET
                                                           #tempSubAck := TRUE;
                                                           #statSwitchCaseHeaderType := #DEFAULT_VALUE_ZERO;
                                                       END_REGION
                                                   #MQTT_MSG_TYPE_UNSUBACK:
                                                       REGION UNSUBACK_PACKET
                                                           #tempUnSubAck := TRUE;
                                                           #statSwitchCaseHeaderType := #DEFAULT_VALUE_ZERO;
                                                       END_REGION
                                                   #MQTT_MSG_TYPE_PINGRESP:
                                                       REGION PINGRESP_PACKET
                                                           #tempPingResp := TRUE;
                                                           #statSwitchCaseHeaderType := #DEFAULT_VALUE_ZERO;
                                                       END_REGION
                                                   #MQTT_MSG_TYPE_PUB_INC_MESSAGE_QoS0, #MQTT_MSG_TYPE_PUB_INC_MESSAGE_QoS1, #MQTT_MSG_TYPE_PUB_INC_MESSAGE_QoS2:
                                                       REGION INC_PUB_PACKET, follow up is WaitForBody
                                                           //we recieved a message on a topic we subscribed to. 
                                                           //ResetBuffer
                                                           #statInternalBufferCount := 0; //set start value
                                                           #statInternalBufferOverflow := FALSE;
                                                           //Evaluate rem. length:
                                                           #tempMultiplier := 1;
                                                           #statRemainingLenOfRecMessage := INT_TO_UDINT(#DEFAULT_VALUE_ZERO);
                                                           #statTotalRemainingMessageLengthSaver := INT_TO_UDINT(#DEFAULT_VALUE_ZERO);

                                                           //when we store only data, we loose info on QoS.. so store for later use.
                                                           IF (#statTrcvHeaderBuffer[1] AND #BIT_MASK_QOS) = INT_TO_BYTE(#MQTT_MSG_TYPE_PUB_INC_MESSAGE_QoS0)
                                                           THEN
                                                               #statRecPackageQoSsaver := #QOS_0;
                                                           ELSIF (#statTrcvHeaderBuffer[1] AND #BIT_MASK_QOS) = INT_TO_BYTE(#MQTT_MSG_TYPE_PUB_INC_MESSAGE_QoS1)
                                                           THEN
                                                               #statRecPackageQoSsaver := #QOS_1;
                                                           ELSIF (#statTrcvHeaderBuffer[1] AND #BIT_MASK_QOS) = INT_TO_BYTE(#MQTT_MSG_TYPE_PUB_INC_MESSAGE_QoS2)
                                                           THEN
                                                               #statRecPackageQoSsaver := #QOS_2;
                                                           ELSIF (#statTrcvHeaderBuffer[1] AND #BIT_MASK_QOS) = INT_TO_BYTE(#MQTT_MSG_TYPE_PUB_INC_MESSAGE_BAD)
                                                           THEN
                                                               //someone send us bad mqtt packet with QoS 1 and 2 to true.
                                                               #statStateTcpMachine := #TCP_ERROR; //close network connection
                                                               #statStatusID := #MQTT_MSG_TYPE_PUB_INC_MESSAGE_BAD;
                                                               #statStatus := #MQTT_ERROR_BADMESSAGE;
                                                           END_IF;

                                                           FOR #statCntOffset := 2 TO 5 DO //calculate rem length of packet according to data provided
                                                               //Goes from Byte 2 in Buffer to Byte 5 in Buffer (max)
                                                               #statRemainingLenOfRecMessage += BYTE_TO_UDINT((#statTrcvHeaderBuffer[#statCntOffset] AND 127)) * #tempMultiplier;
                                                               #tempMultiplier *= 128;
                                                               IF (#tempMultiplier > 128 * 128 * 128)
                                                               THEN//Throw error here // Malformed remain length. might change this
                                                                   ;
                                                               ELSIF ((#statTrcvHeaderBuffer[#statCntOffset] AND 128) = 0)
                                                               THEN //no more data condition, exit loop here
                                                                   //#statRemLenOfIncMes contains remaining length to be expected.
                                                                   EXIT;
                                                               END_IF;
                                                           END_FOR;
                                                           //As we decrease RemLen, we need to save Remaining Len for later.
                                                           #statTotalRemainingMessageLengthSaver := #statRemainingLenOfRecMessage;

                                                           //we might have some message data in the recieve buffer array , so copy to it to internalBuffer;
                                                           IF #statCntOffset < 5 //if its 5, we have 4 byte length identfier(max)
                                                           THEN
                                                               FOR #statInternalBufferCount := 1 TO (5 - #statCntOffset) DO //For 1 to 3 do ...
                                                                   #statInternalBodyBuffer[#statInternalBufferCount] := #statTrcvHeaderBuffer[(#statInternalBufferCount + #statCntOffset)];
                                                                   //Copies data from header buffer to internal body buffer array
                                                               END_FOR;
                                                               //depening on how often we had to extract data
                                                               //rem len <127 means statIOffset=2 so we have 3 byte already of message in internalBuffer
                                                               #statRemainingLenOfRecMessage := #statRemainingLenOfRecMessage - (5 - INT_TO_UINT(#statCntOffset)); //modify rem len  
                                                           END_IF;


                                                           //init for trcvLEN:
                                                           #statTrcvlen := #statRemainingLenOfRecMessage; //up to 1400 bytes
                                                           IF #statTrcvlen > #MAX_TRCV_1400
                                                           THEN
                                                               #statTrcvlen := #MAX_TRCV_1400; //this is max bytes we want to get in one cycle.
                                                           END_IF;
                                                           #statSwitchCaseHeaderType := #DEFAULT_VALUE_ZERO;

                                                           #statStateTrcvMachine := #TRCV_WAIT_FOR_BODY;
                                                       END_REGION
                                                   ELSE  //  ELSE no Valid Header ... maybe data garbage
                                                       FOR #statCnt := 1 TO 5 DO //Clears Buffer
                                                           #statTrcvHeaderBuffer[#statCnt] := INT_TO_BYTE(#DEFAULT_VALUE_ZERO);
                                                       END_FOR;
                                                       #statSwitchCaseHeaderType := #DEFAULT_VALUE_ZERO;
                                               END_CASE;
                                           END_REGION
                                       ELSE
                                           //no new data in this cycle, continue with MQTT Internal StateMachine
                                           //just idle
                                           ;
                                       END_IF;
                                   END_REGION
                               #TRCV_WAIT_FOR_BODY:
                                   REGION WAIT_FOR_BODY
                                       // #statTRCVLEN was set to := #statRemainingLenOfRecMessage or MAX which equals MAX_TRCV_1400
                                       //  #statRemainingLenOfRecMessage holds remaining data length of mqtt message
                                       // check if data arrived:
                                       #statEnableTrcvWatchDogTimer := TRUE;//enable watchdog timer, default is TRCV_WATCHDOG_TIME 2s

                                       IF #instTcpRrcv.BUSY = false AND #instTcpRrcv.NDR = TRUE //we got body 
                                       THEN
                                           #statEnableTrcvWatchDogTimer := FALSE; //Reset Watchdog
                                           #statRemainingLenOfRecMessage := #statRemainingLenOfRecMessage - #instTcpRrcv.RCVD_LEN; //decrease by revieved Len

                                           IF (#statRemainingLenOfRecMessage < #DEFAULT_VALUE_ZERO)//shouldnt happen, just make sure.
                                           THEN
                                               #statRemainingLenOfRecMessage := INT_TO_UDINT(#DEFAULT_VALUE_ZERO);
                                           END_IF;

                                           FOR #tempCnt := 1 TO UDINT_TO_DINT(#instTcpRrcv.RCVD_LEN) // Up to total recieved Bytes
                                           DO
                                               IF (#statInternalBufferCount <= #MAX_INTERNAL_BUFFERLEN) // if it fits in the buffer
                                               THEN
                                                   #statInternalBodyBuffer[#statInternalBufferCount] := #statTrcvMessageBuffer[#tempCnt]; //copy
                                                   #statInternalBufferCount += 1; // increment buffer count by one
                                               ELSE
                                                   #statInternalBufferOverflow := TRUE; //signal overflow;
                                                   EXIT; // leave  LOOP Here, stop copying here
                                               END_IF;
                                           END_FOR;

                                           IF #statRemainingLenOfRecMessage = #DEFAULT_VALUE_ZERO
                                           THEN
                                               //finish #statInternalBodyBuffer is full or complete
                                               #tempReceivedMessage := TRUE; //evaluate in stateMachine #statStateMqttReceive below
                                               #statTrcvlen := INT_TO_UDINT(#DEFAULT_VALUE_ZERO);
                                               #statStateTrcvMachine := #TRCV_WAIT_FOR_HEADER;
                                           ELSE
                                               //continue recieving data untill buffer is full.
                                               #statTrcvlen := #statRemainingLenOfRecMessage; //up to 1400 bytes
                                               IF #statTrcvlen > #MAX_TRCV_1400
                                               THEN
                                                   #statTrcvlen := #MAX_TRCV_1400; //this is max bytes we want to get in one cycle.
                                                   #statStateTrcvMachine := #TRCV_WAIT_FOR_BODY;
                                               END_IF;
                                           END_IF;
                                       ELSE
                                           //else case, if timeout while waiting for TRCV then..
                                           IF #instTrcvWatchDogTimeout.Q
                                               //CHECK FOR TIMEOUT HERE
                                           THEN
                                               #statStateTcpMachine := #TCP_ERROR;
                                               #statStatusID := #TIME_MONITORING_ID;
                                           END_IF;
                                       END_IF;
                                   END_REGION
                               ELSE  // StateMachine section ELSE //generic error?
                                   ;
                           END_CASE;
                       END_REGION
                   END_IF;
               END_REGION


           #TCP_DISCONNECT:
               REGION TCP Disconnect
                   //Start rising edge
                   #instTcpDisconnect.REQ := NOT #instTcpDisconnect.REQ XOR #instTcpDisconnect.BUSY;
                   //no watchdog needed

                   //CALL INSTANCE
                   #instTcpDisconnect(ID := #statTcpConnParam.ConnPara.ID);

                   IF (#instTcpDisconnect.DONE AND #statDisconnect)
                   THEN
                       //Done with success but we had a disconnect
                       #instTcpDisconnect.REQ := false;
                       #statDisconnect := FALSE;
                       #statLastState := #TCP_DISCONNECT;
                       #statStateTcpMachine := #TCP_ERROR; // go to error.
                   ELSIF #instTcpDisconnect.DONE
                   THEN
                       //Done with success 
                       #instTcpDisconnect.REQ := false;
                       #statLastState := #TCP_DISCONNECT;
                       #statStateTcpMachine := #IDLE; // go back to idle.
                   ELSIF (#instTcpDisconnect.ERROR)
                   THEN
                       #statDisconnect := FALSE;
                       #statStatusID := #TCP_DISCONNECT;
                       #instTcpDisconnect.REQ := false;
                       #statStateTcpMachine := #TCP_ERROR;
                   END_IF;
               END_REGION

           #TCP_ERROR:
               REGION TCP Error STATE
                   #statError := true;
                   #statStateTrcvMachine := #TRCV_WAIT_FOR_HEADER;
                   #statStateMqttMachine := #MQTT_DISCONNECTED_STATE; //TCP Broken, so MQTT was disconnected.
                   #statStateMqttJobMachine := #IDLE;
                   #statTcpEstablished := false;
                   #statMqttEstablished := false;
                   #statDone := false;
                   #statEnableTconWatchDogTimer := false;
                   #statEnableTrcvWatchDogTimer := False;
                   CASE #statStatusID OF
                       #TCP_CONNECTING:
                           #statStateTcpMachine := #IDLE;
                           #statStatus := #instTcpConnect.STATUS;
                       #TCP_CONNECTED:
                           IF #statLastState = #TCP_DISCONNECT
                           THEN
                               #statStateTcpMachine := #IDLE;
                           ELSE
                               #statStateTcpMachine := #TCP_DISCONNECT;
                               #statStatus := #instTcpRrcv.STATUS;
                           END_IF;
                       #TCP_DISCONNECT:
                           //pointless for a retry at TDISCON
                           #statStateTcpMachine := #IDLE;
                           #statStatus := #instTcpDisconnect.STATUS;
                       #TIME_MONITORING_ID:
                           #statStateTcpMachine := #TCP_DISCONNECT;
                           #statStatus := TIME_TO_DWORD(IN := #instTconWatchDog.ET);
                       #MQTT_MSG_TYPE_PUB_INC_MESSAGE_BAD:
                           #statStateTcpMachine := #TCP_DISCONNECT;
                           #statStatus := #MQTT_ERROR_BADMESSAGE;
                       ELSE // ELSE CASE StatusID Error
                           ;
                   END_CASE;
               END_REGION
           ELSE // ELSE CASE STATEMACHINE TCP
               ;
       END_CASE;
   END_REGION

   REGION Rising edge detection
       // rising edge detection
       #statEnableOld := #enable;
   END_REGION

   //Bring Statemachine in a definded state, if TCP Connection breaks
   REGION IF TCP breaks go to defined State
       IF #statStateMqttMachine > #IDLE AND
           #statStateTcpMachine <> #TCP_CONNECTED
       THEN
           #statStateMqttMachine := #MQTT_DISCONNECTED_STATE;
           #statStateMqttJobMachine := #IDLE;
           #statStateMqttReceive := #IDLE;
           #instTcpSend.REQ := FALSE;
           #instTcpSendSubscribedMessagesAck.REQ := FALSE;
       END_IF;
   END_REGION

   REGION MQTT KEEPALIVE TIMER
       #instMqttKeepAlivePing(IN := #statEnableMqttKeepAliveTimer,
                              PT := #statMqttKeepAliveTime);

       #instMqttAcknowledgeWatchDog(IN := #statEnableMqttAckWatchDog,
                                    PT := #MQTT_ACK_WATCHDOG_TIME); //default is 10 seconds
       ;
   END_REGION

   // MQTT StateMachine, only Executed if TCP is Connected.
   REGION MQTT STATE MACHINE

       CASE #statStateMqttMachine OF

           #MQTT_DISCONNECTED_STATE:
               REGION DISCONNECTED STATE
                   #statMqttEstablished := false;
                   #statPublishOld := #publishData.publishMessage;
                   #statSubscribeOld := #subscribeToTopic.subscribeToTopic;
                   #statUnsubcribeOld := #subscribeToTopic.unsubscribeFromTopic;
                   #statStateMqttMachine := #MQTT_CONNECT_FLAG_CHECK_STATE;
                   #statStateMqttJobMachine := #IDLE;
                   #statStateMqttReceive := #IDLE;

                   #statEnableMqttKeepAliveTimer := false;
                   #statEnableMqttAckWatchDog := FALSE;
                   #statMqttKeepAliveOff := false;
                   #statPubPacEncoded := false;
                   #statSubPacEncoded := FALSE;
                   #statUnsubPacEncoded := FALSE;
                   #statQoS1decoded := False;
                   #statPingPacEncoded := False;

                   #statPacketID := #DEFAULT_PACKET_ID;
                   // reset packetID
               END_REGION
           #MQTT_CONNECT_FLAG_CHECK_STATE:
               REGION INIT CONNECT STATE
                   #statBusy := true;
                   //validate flags before heading to connect packet!
                   IF #mqttParam.connectFlag.willRetain
                       AND NOT #mqttParam.connectFlag.will
                   THEN
                       #statStateMqttMachine := #MQTT_ERROR_STATE;
                       #statStatusID := #MQTT_CONNECT_FLAG_CHECK_STATE;
                       #statStatus := #MQTT_ERROR_WILL_FLAG;
                   ELSE
                       IF NOT #mqttParam.connectFlag.will
                           AND (#mqttParam.connectFlag.willQoS1 OR #mqttParam.connectFlag.willQoS2)
                       THEN
                           #statStateMqttMachine := #MQTT_ERROR_STATE;
                           #statStatusID := #MQTT_CONNECT_FLAG_CHECK_STATE;
                           #statStatus := #MQTT_ERROR_QOS_FLAG;
                       ELSE
                           IF (#mqttParam.connectFlag.willQoS1
                               AND #mqttParam.connectFlag.willQoS2)
                           THEN
                               #statStateMqttMachine := #MQTT_ERROR_STATE;
                               #statStatusID := #MQTT_CONNECT_FLAG_CHECK_STATE;
                               #statStatus := #MQTT_ERROR_QOS_FLAG;
                           ELSE
                               // all ok, try to connect
                               #statStateMqttMachine := #MQTT_CONNECT_STATE;
                           END_IF;
                       END_IF;
                   END_IF;
                   IF (#mqttParam.keepAlive = #DEFAULT_VALUE_ZERO) // No keepalive was set.
                   THEN
                       #statMqttKeepAliveOff := true;
                   END_IF;

                   IF (#mqttParam.keepAlive < 3) // IF Set to 1 or 2 seconds..
                       AND
                       (#mqttParam.keepAlive > 0)
                   THEN
                       #statStateMqttMachine := #MQTT_ERROR_STATE;
                       #statStatusID := #MQTT_CONNECT_FLAG_CHECK_STATE;
                       #statStatus := #MQTT_ERROR_KEEPALIVE;
                   END_IF;

                   IF (#mqttParam.keepAlive > 2) //if set to more than 2 seconds
                   THEN
                       #statMqttKeepAliveOff := false;
                       //KeepAliveTImer is set to ((Keep Alive converted to seconds) - 2s)
                       #statMqttKeepAliveTime := UINT_TO_TIME((#mqttParam.keepAlive * 1000 - 2000));
                   END_IF;

               END_REGION

           #MQTT_CONNECT_STATE:

               REGION MQTT SEND CONNECT                 
                   //Build Connect packet AND then start TSEND
                   //INIT Buffer Array
                   FILL_BLK(IN:=#EMPTY_CHAR,
                            COUNT:=INT_TO_UINT(#MAX_USER_PW_WILL_LEN)+1,
                            OUT=>#statStringToCharBuffer[0]);

                 //  #statStringToCharBuffer:=0;
                   #statConnectLength := 10 + LEN(IN := #mqttParam.clientIdentifier) + #DEFAULT_TWO_BYTE_LEN;
                   IF #mqttParam.connectFlag.userName
                   THEN
                       #statConnectLength := #statConnectLength + LEN(IN := #mqttParam.userName) + #DEFAULT_TWO_BYTE_LEN;
                   END_IF;
                   IF #mqttParam.connectFlag.password
                   THEN
                       #statConnectLength := #statConnectLength + LEN(IN := #mqttParam.password) + #DEFAULT_TWO_BYTE_LEN;
                   END_IF;
                   IF #mqttParam.connectFlag.will
                   THEN
                       #statConnectLength := #statConnectLength + LEN(IN := #mqttParam.willMessage) + LEN(IN := #mqttParam.willTopic) + (2 * #DEFAULT_TWO_BYTE_LEN);
                   END_IF;
                   //Offset starts with zero
                   #statConnectLengthOffset := #DEFAULT_VALUE_ZERO;
                   //Build Connect Telegram
                   //Fixed Header
                   #statSendBuffer[1] := INT_TO_BYTE(#MQTT_MSG_TYPE_CONNECT);

                   #statSendLength := #statConnectLength;
                   WHILE (#statConnectLength > #DEFAULT_VALUE_ZERO)
                   DO//See MQTT Spec for explanation of this calculation
                       #statConnectEncodedLength := #statConnectLength MOD #CONST_128_CALC;
                       #statConnectLength := #statConnectLength / #CONST_128_CALC;
                       // if there are more data to encode, set the top bit of this byte
                       IF #statConnectLength > #DEFAULT_VALUE_ZERO
                       THEN
                           // Do this and continue while loop
                           //#statConnectEncodedLength :=#statConnectEncodedLength OR 128;
                           #statConnectEncodedLength := WORD_TO_INT(INT_TO_WORD(#statConnectEncodedLength) OR INT_TO_WORD(#CONST_128_CALC));
                           #statSendBuffer[2 + #statConnectLengthOffset] := INT_TO_BYTE(#statConnectEncodedLength);
                           #statConnectLengthOffset += 1;// increment by 1
                       ELSE
                           //do this and leave while loop
                           #statSendBuffer[2 + #statConnectLengthOffset] := INT_TO_BYTE(#statConnectEncodedLength);
                       END_IF;
                   END_WHILE;
                   #statSendLength := #statSendLength + #statConnectLengthOffset;//If offset > zero

                   //Variable Header built telegram
                   //Protocol name
                   #statSendBuffer[3 + #statConnectLengthOffset] := 0;
                   #statSendBuffer[4 + #statConnectLengthOffset] := 4;
                   #statSendBuffer[5 + #statConnectLengthOffset] := CHAR_TO_BYTE('M');
                   #statSendBuffer[6 + #statConnectLengthOffset] := CHAR_TO_BYTE('Q');
                   #statSendBuffer[7 + #statConnectLengthOffset] := CHAR_TO_BYTE('T');
                   #statSendBuffer[8 + #statConnectLengthOffset] := CHAR_TO_BYTE('T');
                   //Protocol Level
                   #statSendBuffer[9 + #statConnectLengthOffset] := INT_TO_BYTE(#MQTT_PROTOCOL_LEVEL);
                   //Connect Flags
                   #statSendBuffer[10 + #statConnectLengthOffset].%X0 := false;
                   #statSendBuffer[10 + #statConnectLengthOffset].%X1 := #mqttParam.connectFlag.cleanSession;
                   #statSendBuffer[10 + #statConnectLengthOffset].%X2 := #mqttParam.connectFlag.will;
                   #statSendBuffer[10 + #statConnectLengthOffset].%X3 := #mqttParam.connectFlag.willQoS1;
                   #statSendBuffer[10 + #statConnectLengthOffset].%X4 := #mqttParam.connectFlag.willQoS2;
                   #statSendBuffer[10 + #statConnectLengthOffset].%X5 := #mqttParam.connectFlag.willRetain;
                   #statSendBuffer[10 + #statConnectLengthOffset].%X6 := #mqttParam.connectFlag.password;
                   #statSendBuffer[10 + #statConnectLengthOffset].%X7 := #mqttParam.connectFlag.userName;
                   //Keep Alive in sec
                   #tempWordForSliceAddress := UINT_TO_WORD(#mqttParam.keepAlive);
                   #statSendBuffer[11 + #statConnectLengthOffset] := #tempWordForSliceAddress.%B1;
                   #statSendBuffer[12 + #statConnectLengthOffset] := #tempWordForSliceAddress.%B0;
                   //Payload
                   //ClientIdentifier
                   #tempLength := INT_TO_WORD(LEN(IN := #mqttParam.clientIdentifier));
                   #statSendBuffer[13 + #statConnectLengthOffset] := #tempLength.%B1;
                   #statSendBuffer[14 + #statConnectLengthOffset] := #tempLength.%B0;

                   Strg_TO_Chars(Strg := #mqttParam.clientIdentifier,
                                 pChars := #DEFAULT_VALUE_ZERO,
                                 Cnt => #tempCountChars,
                                 Chars := #statStringToCharBuffer);

                   FOR #statCnt := #DEFAULT_VALUE_ZERO TO UINT_TO_INT(#tempCountChars - 1) DO
                       #statSendBuffer[15 + #statConnectLengthOffset + #statCnt] := CHAR_TO_BYTE(#statStringToCharBuffer[#statCnt]);
                   END_FOR;
                   #statConnectLengthOffset := #statConnectLengthOffset + DINT_TO_INT(#statCnt);
                   //Will Topic and Will Message
                   IF #mqttParam.connectFlag.will THEN
                       #statCorrectOffset := 0;
                       #tempLength := INT_TO_WORD(LEN(IN := #mqttParam.willTopic));
                       #statSendBuffer[15 + #statConnectLengthOffset] := #tempLength.%B1;
                       #statSendBuffer[16 + #statConnectLengthOffset] := #tempLength.%B0;
                       Strg_TO_Chars(Strg := #mqttParam.willTopic,
                                     pChars := #DEFAULT_VALUE_ZERO,
                                     Cnt => #tempCountChars,
                                     Chars := #statStringToCharBuffer);
                       FOR #statCnt := #DEFAULT_VALUE_ZERO TO UINT_TO_INT(#tempCountChars - 1) DO
                           #statSendBuffer[17 + #statConnectLengthOffset + #statCnt] := CHAR_TO_BYTE(#statStringToCharBuffer[#statCnt]);
                       END_FOR;
                       #statConnectLengthOffset := #statConnectLengthOffset + DINT_TO_INT(#statCnt);

                       #tempLength := INT_TO_WORD(LEN(IN := #mqttParam.willMessage));
                       #statSendBuffer[17 + #statConnectLengthOffset] := #tempLength.%B1;
                       #statSendBuffer[18 + #statConnectLengthOffset] := #tempLength.%B0;
                       Strg_TO_Chars(Strg := #mqttParam.willMessage,
                                     pChars := 0,
                                     Cnt => #tempCountChars,
                                     Chars := #statStringToCharBuffer);
                       FOR #statCnt := 0 TO UINT_TO_INT(#tempCountChars - 1) DO
                           #statSendBuffer[19 + #statConnectLengthOffset + #statCnt] := CHAR_TO_BYTE(#statStringToCharBuffer[#statCnt]);
                       END_FOR;
                       #statConnectLengthOffset := #statConnectLengthOffset + DINT_TO_INT(#statCnt);
                   ELSE
                       #statCorrectOffset := (2 * #DEFAULT_TWO_BYTE_LEN);
                   END_IF;
                   //UserName
                   IF #mqttParam.connectFlag.userName THEN
                       #tempLength := INT_TO_WORD(LEN(IN := #mqttParam.userName));
                       #statSendBuffer[19 + #statConnectLengthOffset - #statCorrectOffset] := #tempLength.%B1;
                       #statSendBuffer[20 + #statConnectLengthOffset - #statCorrectOffset] := #tempLength.%B0;
                       Strg_TO_Chars(Strg := #mqttParam.userName,
                                     pChars := 0,
                                     Cnt => #tempCountChars,
                                     Chars := #statStringToCharBuffer);
                       FOR #statCnt := 0 TO UINT_TO_INT(#tempCountChars - 1) DO
                           #statSendBuffer[21 + #statConnectLengthOffset + #statCnt - #statCorrectOffset] := CHAR_TO_BYTE(#statStringToCharBuffer[#statCnt]);
                       END_FOR;
                       #statConnectLengthOffset := #statConnectLengthOffset + DINT_TO_INT(#statCnt);
                   END_IF;
                   //Password
                   IF #mqttParam.connectFlag.password THEN
                       #tempLength := INT_TO_WORD(LEN(IN := #mqttParam.password));
                       #statSendBuffer[21 + #statConnectLengthOffset - #statCorrectOffset] := #tempLength.%B1;
                       #statSendBuffer[22 + #statConnectLengthOffset - #statCorrectOffset] := #tempLength.%B0;
                       Strg_TO_Chars(Strg := #mqttParam.password,
                                     pChars := 0,
                                     Cnt => #tempCountChars,
                                     Chars := #statStringToCharBuffer);
                       FOR #statCnt := 0 TO UINT_TO_INT(#tempCountChars - 1) DO
                           #statSendBuffer[23 + #statConnectLengthOffset + #statCnt - #statCorrectOffset] := CHAR_TO_BYTE(#statStringToCharBuffer[#statCnt]);
                       END_FOR;
                       #statConnectLengthOffset := #statConnectLengthOffset + DINT_TO_INT(#statCnt);
                   END_IF;

                   //Enable TSEND and start sending data
                   #instTcpSend.REQ := true;
                   #instTcpSend.LEN := INT_TO_UDINT(#statSendLength + #DEFAULT_TWO_BYTE_LEN);

                   IF NOT #statEnableMqttAckWatchDog // if keepAlive was not disabled
                   THEN
                       //KeepAliveTImer is set to (Keep Alive (in s) - 2s)
                       #statEnableMqttAckWatchDog := true; //As long as this is set to true, timers running.
                   END_IF;
                   #statStateMqttMachine := #MQTT_CONNACK_STATE; //go to waiting for conn acknowledge

               END_REGION

           #MQTT_CONNACK_STATE:

               REGION WAIT FOR CONACK
                   //Waiting for the tempConACK from TRCV..

                   IF ((#instTcpSend.DONE) //Check if TSEND went ok last cycle.
                       AND (#instTcpSend.BUSY = false))
                   THEN
                       #instTcpSend.REQ := false; // reset send trigger
                       //Delete Send Buffer
                       FOR #statCnt := 1 TO (#statSendLength + #DEFAULT_TWO_BYTE_LEN) DO
                           #statSendBuffer[#statCnt] := 0; //Clears buffer;
                       END_FOR;
                   ELSIF #instTcpSend.ERROR
                   THEN // Tsend error occured
                       #statEnableMqttAckWatchDog := False;
                       #statStatusID := #MQTT_CONNECT_STATE;
                       #instTcpSend.REQ := false;
                       #statStateMqttMachine := #MQTT_ERROR_STATE;
                   END_IF;

                   //recieved CONACK Package
                   IF #tempConAck THEN
                       #statEnableMqttAckWatchDog := False;
                       //We have now data in TRCVHeaderBuffer(3Byte properly)
                       IF (#statTrcvHeaderBuffer[2] AND #BIT_MASK_LOWBITS) = 2 //remainng Length must be 2;
                       THEN //
                           //byte one is 0000 000X where X is if Session was set // so depending on clean session or not we evaluate answer of server
                           IF (#mqttParam.connectFlag.cleanSession = FALSE AND (#statTrcvHeaderBuffer[3] AND #BIT_MASK_LOWBITS) = INT_TO_BYTE(#MQTT_CONACK_FLAG_SP))
                               OR (#mqttParam.connectFlag.cleanSession = TRUE AND (#statTrcvHeaderBuffer[3] AND 16#00) = 0)
                           THEN
                               //VALID Answer, check code
                               IF (#statTrcvHeaderBuffer[4] = INT_TO_BYTE(#MQTT_CONNACK_ACCEPTED))
                               THEN
                                   //VALID
                                   #statStateMqttMachine := #MQTT_CONNECTED_STATE;
                                   #statMqttEstablished := true;
                                   #statBusy := false;
                                   #statStateMqttJobMachine := #IDLE;
                               ELSE
                                   //NOT VALID e.g we have an error
                                   #statStateMqttMachine := #MQTT_ERROR_STATE;
                                   #statStatus := #statTrcvHeaderBuffer[4]; // maybe we got an error message in buffer
                                   #statStatusID := #MQTT_CONNACK_STATE;
                               END_IF;
                           ELSE
                               //NOT VALID
                               //Signal error and go to error State.
                               #statStateMqttMachine := #MQTT_ERROR_STATE;
                               #statStatus := #statTrcvHeaderBuffer[3]; // Clean Session Mismatch ERROR
                               #statStatusID := #MQTT_CONNACK_STATE;
                           END_IF;
                       ELSE // We got a CONNACK paket, but remaining length was not 2 (Error)
                           //NOT VALID
                           //Signal error and go to error State.
                           #statStateMqttMachine := #MQTT_ERROR_STATE;
                           #statStatus := #statTrcvHeaderBuffer[2];
                           #statStatusID := #MQTT_BAD_ID;
                           // After Error state we go to #MQTT_DISCONNECTED AND Disconnect TCP.
                       END_IF;
                       // keepalive triggered, no reaction from server. must close network connection.
                   ELSIF #instMqttAcknowledgeWatchDog.Q
                   THEN
                       #statStateMqttMachine := #MQTT_ERROR_STATE;
                       #statStatus := #MQTT_ERROR_KEEPALIVE;
                       #statStatusID := #MQTT_TIMEOUT_ID; // we go to time out error state and then close TCP.
                       #statEnableMqttAckWatchDog := FALSE; // we can shut down timer now.
                   END_IF;

               END_REGION

           #MQTT_CONNECTED_STATE:

               REGION MQTT CONNECTED wait for input  
                   REGION CHECK FOR JOBS
                       REGION IF PING packet Timer expired
                           // we are Connected, first check if we have to send keepAlive
                           IF (#instMqttKeepAlivePing.Q) // Timer expired
                               AND (#statStateMqttJobMachine = #IDLE) // and we have no job
                               AND (NOT #statMqttKeepAliveOff) // And keepalive is not off
                           THEN
                               #statStateMqttJobMachine := #MQTT_PING;
                               #statBusy := true;
                               #statEnableMqttKeepAliveTimer := false; //reset timer edge // will be set to true, when ping complete and back to IDLE state..
                           END_IF;
                       END_REGION

                       REGION IFPublish
                           IF #publishData.publishMessage
                               AND NOT #subscribeToTopic.subscribeToTopic
                               AND NOT #subscribeToTopic.unsubscribeFromTopic
                               AND NOT #statPublishOld
                               AND (#statStateMqttJobMachine = #IDLE)
                           THEN
                               #statBusy := true;
                               #statStateMqttJobMachine := #MQTT_PUBLISH_STATE;
                               #statEnableMqttKeepAliveTimer := false; //disable PingTimer
                               IF #statPacketID < #MAX_INT
                               THEN
                                   #statPacketID += 1; // increment
                               ELSE
                                   #statPacketID := #DEFAULT_PACKET_ID;
                               END_IF;
                           END_IF;
                           #statPublishOld := #publishData.publishMessage;
                       END_REGION

                       REGION IFSubscribe
                           IF #subscribeToTopic.subscribeToTopic
                               AND NOT #publishData.publishMessage
                               AND NOT #subscribeToTopic.unsubscribeFromTopic
                               AND NOT #statSubscribeOld
                               AND (#statStateMqttJobMachine = #IDLE)

                           THEN
                               #statBusy := true;
                               #statStateMqttJobMachine := #MQTT_SUBSCRIBE_STATE;
                               #statEnableMqttKeepAliveTimer := false; //disable PingTimer

                               IF #statPacketID < #MAX_INT
                               THEN
                                   #statPacketID += 1;
                               ELSE
                                   #statPacketID := #DEFAULT_PACKET_ID;
                               END_IF;

                           END_IF;
                           #statSubscribeOld := #subscribeToTopic.subscribeToTopic;
                       END_REGION

                       REGION IFUnsubscribe
                           IF #subscribeToTopic.unsubscribeFromTopic
                               AND NOT #publishData.publishMessage
                               AND NOT #subscribeToTopic.subscribeToTopic
                               AND NOT #statUnsubcribeOld
                               AND (#statStateMqttJobMachine = #IDLE)
                           THEN
                               #statBusy := true;
                               #statStateMqttJobMachine := #MQTT_UNSUBSCRIBE_STATE;
                               #statEnableMqttKeepAliveTimer := false;

                               IF #statPacketID < #MAX_INT
                               THEN
                                   #statPacketID += 1;
                               ELSE
                                   #statPacketID := #DEFAULT_PACKET_ID;
                               END_IF;
                           END_IF;
                           #statUnsubcribeOld := #subscribeToTopic.unsubscribeFromTopic;
                       END_REGION
                   END_REGION

                   REGION CHECK_IF_RECEIVED MESSAGE on SUBSCRIPTION
                       //we got data this cycle,
                       //its consistent  in the statInternalBodyBuffer Array
                       //and statQos is set
                       //Decide, which QoS Procedure we have to do
                       IF #tempReceivedMessage AND #statStateMqttReceive = #IDLE AND #statRecPackageQoSsaver = #QOS_0
                       THEN
                           #statStateMqttReceive := #MQTT_RECEIVED_QOS0_STATE;
                       ELSIF #tempReceivedMessage AND #statStateMqttReceive = #IDLE AND #statRecPackageQoSsaver = #QOS_1
                       THEN
                           #statStateMqttReceive := #MQTT_RECEIVED_QOS1_STATE;
                       ELSIF #tempReceivedMessage AND #statStateMqttReceive = #IDLE AND #statRecPackageQoSsaver = #QOS_2
                       THEN
                           #statStateMqttReceive := #MQTT_RECEIVED_QOS2_STATE;
                       END_IF;

                   END_REGION

                   REGION Receive Message State Machine
                       //     Subscribed Telegramm Data to Message Output and send Response
                       CASE #statStateMqttReceive OF
                           #IDLE:
                               REGION IDLE
                                   #subscriptionMessage.newMessageRecieved := FALSE; // Reset Output and wait for new incoming messages
                                   #subscriptionMessage.messageInvalid := false;
                                   #statQoS1decoded := FALSE;
                               END_REGION
                           #MQTT_RECEIVED_QOS0_STATE:
                               REGION Recieved QoS0 Message
                                   // QoS 0 = no Response necessary  //Receive Topic/Message QoS0    

                                   //Reset Output, before filling with valid data:
                                   #subscriptionMessage.receivedMessageData := #EMPTY;
                                   #subscriptionMessage.receivingTopic := #EMPTY;

                                   //   The internal buffer only holds the message,
                                   //   no remaining length of whole message,
                                   //    that why we have  #statMesRemLengthSaver
                                   //    only rem topic length is in the buffer

                                   //topic len; byte1&2.

                                   #tempWordForSliceAddress.%B1 := #statInternalBodyBuffer[1];
                                   #tempWordForSliceAddress.%B0 := #statInternalBodyBuffer[2];//max 65 000 bytes

                                   #tempRecPubTopicLength := WORD_TO_UINT(#tempWordForSliceAddress);

                                   IF #tempRecPubTopicLength + #TOPIC_LEN_INFO > #MAX_INTERNAL_BUFFERLEN
                                   THEN
                                       #tempRecPubTopicLength := UDINT_TO_UINT(#MAX_INTERNAL_BUFFERLEN); // topic to long;
                                   END_IF;

                                   FOR #tempCnt := 1 TO UINT_TO_DINT(#tempRecPubTopicLength)
                                   DO
                                       IF #tempCnt < MAX_LEN(#subscriptionMessage.receivingTopic)
                                       THEN
                                           #subscriptionMessage.receivingTopic[#tempCnt] := BYTE_TO_WCHAR(#statInternalBodyBuffer[#TOPIC_LEN_INFO + #tempCnt]);
                                       ELSE
                                           #subscriptionMessage.messageInvalid := TRUE;
                                           EXIT;
                                       END_IF;
                                   END_FOR;

                                   IF (#statTotalRemainingMessageLengthSaver > #MAX_INTERNAL_BUFFERLEN)
                                   THEN
                                       #statTotalRemainingMessageLengthSaver := #MAX_INTERNAL_BUFFERLEN; //Message len too long
                                   END_IF;

                                   IF ((#tempRecPubTopicLength + #TOPIC_LEN_INFO) < #MAX_INTERNAL_BUFFERLEN)//len +2byte len info , if topic is longer and buffer is full, skip this
                                   THEN
                                       FOR #tempCnt := 1 TO UDINT_TO_DINT(#statTotalRemainingMessageLengthSaver - #TOPIC_LEN_INFO - #tempRecPubTopicLength)
                                       DO
                                           IF #tempCnt < MAX_LEN(#subscriptionMessage.receivedMessageData)
                                           THEN
                                               #subscriptionMessage.receivedMessageData[#tempCnt] := BYTE_TO_WCHAR(#statInternalBodyBuffer[#TOPIC_LEN_INFO + #tempRecPubTopicLength + #tempCnt]);
                                           ELSE
                                               #subscriptionMessage.messageInvalid := TRUE;
                                               EXIT;
                                           END_IF;
                                       END_FOR;
                                   END_IF;

                                   IF #statInternalBufferOverflow THEN
                                       #subscriptionMessage.messageInvalid := TRUE;
                                       #statInternalBufferOverflow := false;
                                   END_IF;
                                   #subscriptionMessage.newMessageRecieved := TRUE; //signal that new data is available
                                   #statStateMqttReceive := #IDLE; //reset to idle and wait for new data.
                               END_REGION

                           #MQTT_RECEIVED_QOS1_STATE:
                               REGION Recieved QoS1 Message
                                   //Receive Topic/Message QoS1 and send Publish Ack

                                   //Reset Output, before filling with valid data:
                                   #subscriptionMessage.receivedMessageData := #EMPTY;
                                   #subscriptionMessage.receivingTopic := #EMPTY;

                                   //   The internal buffer only holds the message,
                                   //   no remaining length of whole message,
                                   //    that why we have  #statMesRemLengthSaver
                                   //    only rem topic length is in the buffer
                                   IF NOT #statQoS1decoded THEN
                                       //topic len; byte1&2.

                                       #tempWordForSliceAddress.%B1 := #statInternalBodyBuffer[1];
                                       #tempWordForSliceAddress.%B0 := #statInternalBodyBuffer[2];//max 65 000

                                       #tempRecPubTopicLength := WORD_TO_UINT(#tempWordForSliceAddress);

                                       IF #tempRecPubTopicLength + #TOPIC_LEN_INFO > #MAX_INTERNAL_BUFFERLEN  // check, if topic too long we only need  whats in the buffer
                                       THEN
                                           #tempRecPubTopicLength := UDINT_TO_UINT(#MAX_INTERNAL_BUFFERLEN);
                                       END_IF;

                                       IF (#tempRecPubTopicLength < #MAX_INTERNAL_BUFFERLEN - INT_TO_UDINT(#DEFAULT_TWO_BYTE_LEN)) // check, if topic too long we might lost PacketID.
                                       THEN
                                           #statPacketID2.%B1 := #statInternalBodyBuffer[3 + #tempRecPubTopicLength];
                                           #statPacketID2.%B0 := #statInternalBodyBuffer[4 + #tempRecPubTopicLength];
                                       END_IF;

                                       FOR #tempCnt := 1 TO UINT_TO_DINT(#tempRecPubTopicLength)
                                       DO
                                           IF #tempCnt < MAX_LEN(#subscriptionMessage.receivingTopic)//put everything that fits from buffer to topic output
                                           THEN
                                               #subscriptionMessage.receivingTopic[#tempCnt] := BYTE_TO_WCHAR(#statInternalBodyBuffer[#TOPIC_LEN_INFO + #tempCnt]);
                                           ELSE
                                               #subscriptionMessage.messageInvalid := TRUE;
                                               EXIT;
                                           END_IF;
                                       END_FOR;

                                       IF (#statTotalRemainingMessageLengthSaver > #MAX_INTERNAL_BUFFERLEN)//if there is a huge payload exceeding internal buffer.
                                       THEN
                                           #statTotalRemainingMessageLengthSaver := #MAX_INTERNAL_BUFFERLEN;
                                       END_IF;

                                       IF (#tempRecPubTopicLength + #TOPIC_LEN_INFO + INT_TO_UINT(#DEFAULT_TWO_BYTE_LEN) < #MAX_INTERNAL_BUFFERLEN)//len +2byte len info +2byte packetID
                                       THEN
                                           FOR #tempCnt := 1 TO UDINT_TO_DINT(#statTotalRemainingMessageLengthSaver - #TOPIC_LEN_INFO - #tempRecPubTopicLength - INT_TO_UINT(#DEFAULT_TWO_BYTE_LEN))
                                           DO
                                               IF #tempCnt < MAX_LEN(#subscriptionMessage.receivedMessageData)//put everything that fits to output message
                                               THEN
                                                   #subscriptionMessage.receivedMessageData[#tempCnt] := BYTE_TO_WCHAR(#statInternalBodyBuffer[#TOPIC_LEN_INFO + INT_TO_UINT(#DEFAULT_TWO_BYTE_LEN) + #tempRecPubTopicLength + #tempCnt]);
                                               ELSE
                                                   #subscriptionMessage.messageInvalid := TRUE;
                                                   EXIT;
                                               END_IF;
                                           END_FOR;
                                       END_IF;

                                       IF #statInternalBufferOverflow THEN
                                           #subscriptionMessage.messageInvalid := TRUE;
                                           #statInternalBufferOverflow := false;
                                       END_IF;

                                       //PUBACK - Send Publish acknowledge packet
                                       //fixed Header
                                       #statSendBufferSubscribePacketAckn[1] := INT_TO_BYTE(#MQTT_MSG_TYPE_PUBACK);
                                       #statSendBufferSubscribePacketAckn[2] := INT_TO_BYTE(#DEFAULT_TWO_BYTE_LEN);

                                       //Variable Header
                                       #statSendBufferSubscribePacketAckn[3] := #statPacketID2.%B1; //if buffer overflow, this is a guessing game
                                       #statSendBufferSubscribePacketAckn[4] := #statPacketID2.%B0;
                                       #instTcpSendSubscribedMessagesAck.LEN := INT_TO_UDINT(2 * (#DEFAULT_TWO_BYTE_LEN));

                                       #subscriptionMessage.newMessageRecieved := TRUE; //signal that new data is available
                                       #statQoS1decoded := true;
                                   ELSE
                                       //ensure its only valid for 1 cycle
                                       #subscriptionMessage.newMessageRecieved := FALSE;
                                       #subscriptionMessage.messageInvalid := FALSE;

                                   END_IF;

